// TIA Portal V15.1 export
// export: Created 2024-06-21T08:41:08.920552Z, ExportSetting WithDefaults, DisplayName Totally Integrated Automation Portal, DisplayVersion V15.1 Update 5, DisplayName TIA Portal Openness, DisplayVersion V15.1 Update 5, DisplayName SINAMICS Startdrive Advanced, DisplayVersion V15.1, DisplayName G130, G150, S120, S150, SINAMICS MV, S210, DisplayVersion V15.1, DisplayName G110M, G120, G120C, G120D, G120P, DisplayVersion V15.1, DisplayName STEP 7 Professional, DisplayVersion V15.1 Update 5, DisplayName STEP 7 Safety, DisplayVersion V15.1, DisplayName WinCC Professional, DisplayVersion V15.1 Update 5, DisplayName SIMATIC Visualization Architect, DisplayVersion V15.1
FUNCTION "LGBJoyStick-Config" : Void   // FC6647, FBD
TITLE = LGBJoyStick-Config
{ S7_Optimized_Access := 'TRUE' }
AUTHOR : VCG
VERSION : 0.1
// ============================================================================
// Handles the LJoyStick Config
// ============================================================================
// stored: AutoNumber false, IsIECCheckEnabled false, SetENOAutomatically False, UDAEnableTagReadback false
   VAR_INPUT
      C_BtnMiddleUsed : Bool;   // Button Middle Used
      C_BtnUpUsed : Bool;   // Button Up Used
      C_BtnRightUsed : Bool;   // Button Right Used
      C_BtnDownUsed : Bool;   // Button Down Used
      C_BtnLeftUsed : Bool;   // Button Left Used
      C_BtnExternalUsed : Bool;   // External Buttons Used
      C_BtnUpBlock : Bool;   // Button Up is a Block (0 = Force, 1 = Block)
      C_BtnRightBlock : Bool;   // Button Right is a Block (0 = Force, 1 = Block)
      C_BtnDownBlock : Bool;   // Button Down is a Block (0 = Force, 1 = Block)
      C_BtnLeftBlock : Bool;   // Button Left is a Block (0 = Force, 1 = Block)
      C_BtnUpDesc : String;   // Description button Up
      C_BtnRightDesc : String;   // Description button Right
      C_BtnDownDesc : String;   // Description button Down
      C_BtnLeftDesc : String;   // Description button Left
      C_BtnExternalDesc : String;   // Description External Buttons
   END_VAR
   VAR_IN_OUT
      IO_Config : "JoyStickConfig";   // Config
   END_VAR
BEGIN

REGION Network 1: **** 1 - Inputs **** Move Config
   // Move Config
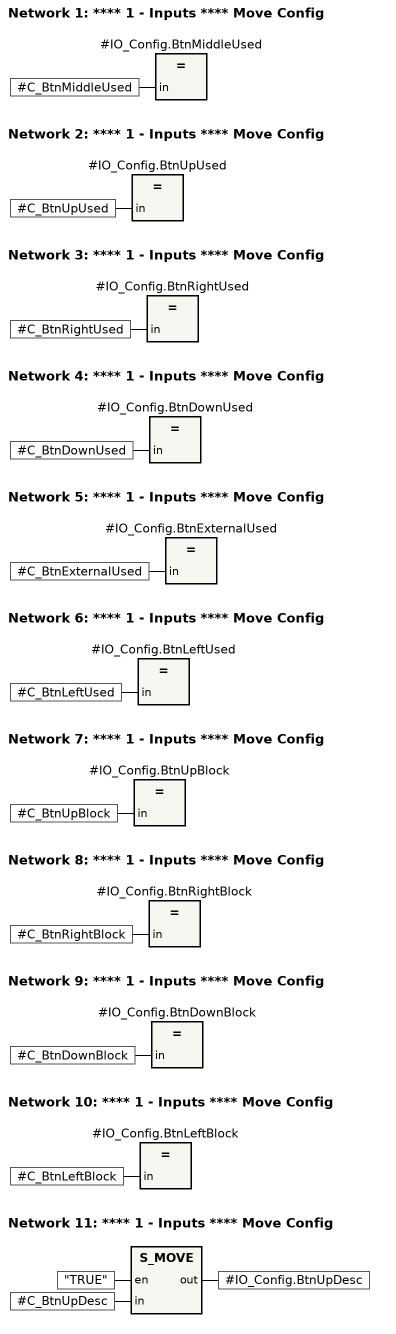
   #IO_Config.BtnMiddleUsed := #C_BtnMiddleUsed;
END_REGION

REGION Network 2: **** 1 - Inputs **** Move Config
   // Move Config
   #IO_Config.BtnUpUsed := #C_BtnUpUsed;
END_REGION

REGION Network 3: **** 1 - Inputs **** Move Config
   // Move Config
   #IO_Config.BtnRightUsed := #C_BtnRightUsed;
END_REGION

REGION Network 4: **** 1 - Inputs **** Move Config
   // Move Config
   #IO_Config.BtnDownUsed := #C_BtnDownUsed;
END_REGION

REGION Network 5: **** 1 - Inputs **** Move Config
   // Move Config
   #IO_Config.BtnExternalUsed := #C_BtnExternalUsed;
END_REGION

REGION Network 6: **** 1 - Inputs **** Move Config
   // Move Config
   #IO_Config.BtnLeftUsed := #C_BtnLeftUsed;
END_REGION

REGION Network 7: **** 1 - Inputs **** Move Config
   // Move Config
   #IO_Config.BtnUpBlock := #C_BtnUpBlock;
END_REGION

REGION Network 8: **** 1 - Inputs **** Move Config
   // Move Config
   #IO_Config.BtnRightBlock := #C_BtnRightBlock;
END_REGION

REGION Network 9: **** 1 - Inputs **** Move Config
   // Move Config
   #IO_Config.BtnDownBlock := #C_BtnDownBlock;
END_REGION

REGION Network 10: **** 1 - Inputs **** Move Config
   // Move Config
   #IO_Config.BtnLeftBlock := #C_BtnLeftBlock;
END_REGION

REGION Network 11: **** 1 - Inputs **** Move Config
   // Move Config
   IF "TRUE" THEN #IO_Config.BtnUpDesc := #C_BtnUpDesc; END_IF;
END_REGION

REGION Network 12: **** 1 - Inputs **** Move Config
   // Move Config
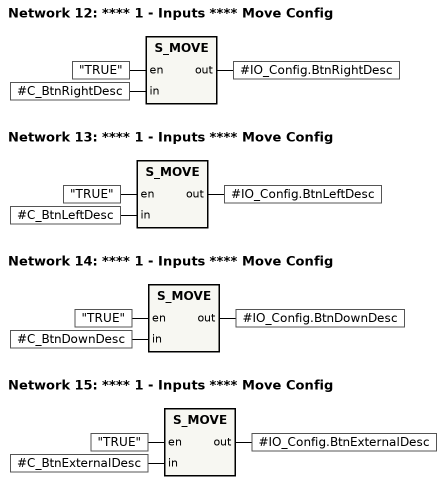
   IF "TRUE" THEN #IO_Config.BtnRightDesc := #C_BtnRightDesc; END_IF;
END_REGION

REGION Network 13: **** 1 - Inputs **** Move Config
   // Move Config
   IF "TRUE" THEN #IO_Config.BtnLeftDesc := #C_BtnLeftDesc; END_IF;
END_REGION

REGION Network 14: **** 1 - Inputs **** Move Config
   // Move Config
   IF "TRUE" THEN #IO_Config.BtnDownDesc := #C_BtnDownDesc; END_IF;
END_REGION

REGION Network 15: **** 1 - Inputs **** Move Config
   // Move Config
   IF "TRUE" THEN #IO_Config.BtnExternalDesc := #C_BtnExternalDesc; END_IF;
END_REGION
END_FUNCTION
